// TIA Portal V17 export
// export: Created 2024-08-20T13:26:09.4945739Z, ExportSetting WithDefaults, DisplayName Totally Integrated Automation Portal, DisplayVersion V17 Update 4, DisplayName TIA Portal Openness, DisplayVersion V17 Update 4, DisplayName TIA Portal Version Control Interface, DisplayVersion V17, DisplayName STEP 7 Professional, DisplayVersion V17 Update 4, DisplayName STEP 7 Safety, DisplayVersion V17, DisplayName WinCC Advanced, DisplayVersion V17 Update 4
DATA_BLOCK "ALARMES"   // DB301
{ S7_Optimized_Access := 'TRUE' }
VERSION : 0.1
// stored: AutoNumber false, DBAccessibleFromOPCUA true, IsOnlyStoredInLoadMemory false, IsRetainMemResEnabled false, IsWriteProtectedInAS false, MemoryReserve 100
   VAR
      "CCM-02-EA-P100-YFC" : Bool;   // Falha de comunicação com medidor do CCM1
      "CCM-02-EB-P100-YFC" : Bool;   // Falha de comunicação com medidor do CCM2
      "LIT_001-YHH" : Bool;   // Alarme de nível muito alto do tanque água bruta
      "LIT_001-YH" : Bool;   // Alarme de nível alto do tanque água bruta
      "LIT_001-YL" : Bool;   // Alarme de nível baixo do tanque água bruta
      "LIT_001-YLL" : Bool;   // Alarme de nível muito baixo do tanque água bruta
      "LIT_001-YFS" : Bool;   // Transmissor de nível do tanque água bruta com falha de sinal
      "LIT_001-YHHH" : Bool;   // Alarme de nível muito alto - desliga CAB e lavagem peneira
      "CAB-PT-015-YH" : Bool;
      "CAB-PT-015-YFS" : Bool;
      "MB-03-YIP" : Bool;   // MB-03 com intervalo entre partidas
      "MB-02-YIP" : Bool;   // MB-02 com intervalo entre partidas
      "MB-01-YIP" : Bool;   // MB-01 com intervalo entre partidas
   END_VAR
BEGIN
END_DATA_BLOCK
